# B&R Automation Studio project VirtualModellingOfEngine
Automation Studio 4.5.2.102

## Configuration Config1

CPU 4PP065.0351-P74, AutomationRuntime D4.52, Build 4.1.2, Vc V4.52.0

### Task classes (Cpu.sw)
```
Cyclic#4:
  Program <- Program.prg
Libraries: Library
```

### Hardware
```
4PP065_0351_P74 : 4PP065.0351-P74 v1.0.4.0
  Connector IF5:
    ActivateDevice = 1
  ConfigurationID = Lab1_2_Config1
  Simulation = 1
  KeyMappingFile = VC\4PP065_0351_P74.dis
```

## Logical view

### Program Logical/Program (ANSIC)

#### Main.c - Init, cyclic, exit code
```c
#include <bur/plctypes.h>

#ifdef _DEFAULT_INCLUDES
	#include <AsDefault.h>
#endif

REAL count = 0;

void _INIT ProgramInit(void)
{
	speed = 0;
	fb_motor.dt = 0.002;
	fb_motor.ke = 2;
	fb_motor.Tm = 0.04;

	fb_regulator.dt = 0.002;
	fb_regulator.e = speed - fb_motor.w;
	fb_regulator.iyOld = 0;
	fb_regulator.max_abs_value = 5;
	fb_regulator.k_i = 20;
	fb_regulator.k_p = 8;

	fb_secondMotor.dt = 0.002;
	fb_secondMotor.ke = 2;
	fb_secondMotor.Tm = 0.04;

	enable = 1;
}

void _CYCLIC ProgramCyclic(void)
{
	if(enable == 1)
	{
		count += 100;
		if((count >= 10000) && (count <= 30000))
		{
			speed = 3;
		}
		else
		{
			speed = 0;
		}

		// motor with regulator
		fb_regulator.e = speed - fb_motor.w;
		FB_regulator(&fb_regulator);
		fb_motor.u = fb_regulator.u;
		FB_Motor(&fb_motor);

		// motor without regulator
		fb_secondMotor.u = speed;
		FB_SecondMotor(&fb_secondMotor);
	}
}

void _EXIT ProgramExit(void)
{

}
```

#### Variables.var - Local variables
```iecst
VAR
	fb_secondMotor : FB_SecondMotor;
	fb_regulator : FB_regulator;
	fb_motor : FB_Motor;
	speed : REAL;
	enable : BOOL;
END_VAR
```

### Library Logical/Library (ANSIC)

#### Library.fun - Exported functions and function blocks
```iecst
{REDUND_ERROR} {REDUND_UNREPLICABLE} FUNCTION_BLOCK FB_regulator (*TODO: Add your comment here*) (*$GROUP=User,$CAT=User,$GROUPICON=User.png,$CATICON=User.png*)
	VAR_INPUT
		e : {REDUND_UNREPLICABLE} REAL;
	END_VAR
	VAR_OUTPUT
		u : {REDUND_UNREPLICABLE} REAL;
	END_VAR
	VAR
		k_p : {REDUND_UNREPLICABLE} REAL;
		k_i : {REDUND_UNREPLICABLE} REAL;
		integrator : {REDUND_UNREPLICABLE} FB_Integrator;
		iyOld : {REDUND_UNREPLICABLE} REAL;
		max_abs_value : {REDUND_UNREPLICABLE} REAL;
		dt : {REDUND_UNREPLICABLE} REAL;
	END_VAR
END_FUNCTION_BLOCK

{REDUND_ERROR} {REDUND_UNREPLICABLE} FUNCTION_BLOCK FB_Integrator (*TODO: Add your comment here*) (*$GROUP=User,$CAT=User,$GROUPICON=User.png,$CATICON=User.png*)
	VAR_INPUT
		in : {REDUND_UNREPLICABLE} REAL;
	END_VAR
	VAR_OUTPUT
		out : {REDUND_UNREPLICABLE} REAL;
	END_VAR
	VAR
		dt : {REDUND_UNREPLICABLE} REAL;
	END_VAR
END_FUNCTION_BLOCK

{REDUND_ERROR} FUNCTION_BLOCK FB_Motor (*TODO: Add your comment here*) (*$GROUP=User,$CAT=User,$GROUPICON=User.png,$CATICON=User.png*)
	VAR_INPUT
		u : {REDUND_UNREPLICABLE} REAL;
	END_VAR
	VAR_OUTPUT
		w : REAL;
		phi : REAL;
	END_VAR
	VAR
		integrator : FB_Integrator;
		Tm : REAL;
		ke : REAL;
		dt : REAL;
	END_VAR
END_FUNCTION_BLOCK

{REDUND_ERROR} FUNCTION_BLOCK FB_SecondMotor (*TODO: Add your comment here*) (*$GROUP=User,$CAT=User,$GROUPICON=User.png,$CATICON=User.png*)
	VAR_INPUT
		u : {REDUND_UNREPLICABLE} REAL;
	END_VAR
	VAR_OUTPUT
		w : REAL;
		phi : REAL;
	END_VAR
	VAR
		integrator : FB_SecondIntegrator;
		Tm : REAL;
		ke : REAL;
		dt : REAL;
	END_VAR
END_FUNCTION_BLOCK

{REDUND_ERROR} {REDUND_UNREPLICABLE} FUNCTION_BLOCK FB_SecondIntegrator (*TODO: Add your comment here*) (*$GROUP=User,$CAT=User,$GROUPICON=User.png,$CATICON=User.png*)
	VAR_INPUT
		in : {REDUND_UNREPLICABLE} REAL;
	END_VAR
	VAR_OUTPUT
		out : {REDUND_UNREPLICABLE} REAL;
	END_VAR
	VAR
		dt : {REDUND_UNREPLICABLE} REAL;
	END_VAR
END_FUNCTION_BLOCK
```

#### FB_regulator.c
```c
#include <bur/plctypes.h>
#ifdef __cplusplus
	extern "C"
	{
#endif
	#include "Library.h"
#ifdef __cplusplus
	};
#endif
/* TODO: Add your comment here */
void FB_regulator(struct FB_regulator* inst)
{
	/*TODO: Add your code here*/
	//Building regulator's structure

	REAL firstPath = 0;		// the one of the scheme's parts
	REAL secondPath = 0;	// the another of the scheme's parts
	if((inst->e*inst->k_p) < (inst->max_abs_value))
	{
		firstPath = inst->e*inst->k_p;
	}
	else
	{
		firstPath = inst->max_abs_value;
	}

	inst->integrator.in = inst->e*inst->k_i*inst->dt + inst->iyOld;
	FB_Integrator(&(inst->integrator));
	secondPath = inst->integrator.out;
	// add into function the antiAccumulationPart
	if((firstPath + secondPath) < (inst->max_abs_value))
		{
			inst->u = (firstPath + secondPath);
		}
	else
		{
			inst->u = inst->max_abs_value;
		}
	 inst->iyOld = inst->u - (firstPath + secondPath);

}
```

#### FB_Integrator.c
```c
#include <bur/plctypes.h>
#ifdef __cplusplus
	extern "C"
	{
#endif
	#include "Library.h"
#ifdef __cplusplus
	};
#endif
/* TODO: Add your comment here */
void FB_Integrator(struct FB_Integrator* inst)
{
	/*TODO: Add your code here*/
	//Building integrator structure
	inst->out = inst->out + inst->in;
}
```

#### FB_Motor.c
```c
#include <bur/plctypes.h>
#ifdef __cplusplus
	extern "C"
	{
#endif
	#include "Library.h"
#ifdef __cplusplus
	};
#endif
/* TODO: Add your comment here */
void FB_Motor(struct FB_Motor* inst)
{
	/*TODO: Add your code here*/
	//Building motor structure
	//for w output
	inst->integrator.in = ((1/(inst->ke))*(inst->u)-(inst->w))*((inst->dt)/(inst->Tm));
	FB_Integrator(&(inst->integrator));
	inst->w = inst->integrator.out;
	//for phi output
	inst->integrator.in = (inst->w)*(inst->dt);
	FB_Integrator(&(inst->integrator));
	inst->phi = inst->integrator.out;
}
```

#### FB_SecondMotor.c
```c
#include <bur/plctypes.h>
#ifdef __cplusplus
	extern "C"
	{
#endif
	#include "Library.h"
#ifdef __cplusplus
	};
#endif
/* TODO: Add your comment here */
void FB_SecondMotor(struct FB_SecondMotor* inst)
{
	/*TODO: Add your code here*/
	inst->integrator.in = ((1/(inst->ke))*(inst->u)-(inst->w))*((inst->dt)/(inst->Tm));
	FB_Integrator(&(inst->integrator));
	inst->w = inst->integrator.out;
	//for phi output
	inst->integrator.in = (inst->w)*(inst->dt);
	FB_Integrator(&(inst->integrator));
	inst->phi = inst->integrator.out;
}
```

#### FB_SecondIntegrator.c
```c
#include <bur/plctypes.h>
#ifdef __cplusplus
	extern "C"
	{
#endif
	#include "Library.h"
#ifdef __cplusplus
	};
#endif
/* TODO: Add your comment here */
void FB_SecondIntegrator(struct FB_SecondIntegrator* inst)
{
	/*TODO: Add your code here*/
	//Building integrator structure
	inst->out = inst->out + inst->in;
}
```

Listed in the project but not available here: Logical/Global.typ, Logical/Global.var, Logical/Libraries, Logical/Program/Types.typ, Logical/Library/Types.typ, Logical/Library/Constants.var
